// Implicitly generated code : DO NOT EDIT
FUNCTION CheckBounds : DINT
VAR_INPUT
	index, lower, upper: DINT;
END_VAR

// Implicitly generated code : Only an Implementation suggestion
{noflow}
IF  index < lower THEN
	CheckBounds := lower;
ELSIF  index > upper THEN
	CheckBounds := upper;
ELSE  
	CheckBounds := index;
END_IF
{flow}

END_FUNCTION

(* stored: Version 1.1.0.1, ProductVersion 3.1.4024.0
   POU CheckBounds: Id {4aa71e58-8a22-49e2-8b69-c56cbe34a862}, SpecialFunc CheckBounds *)
